// TIA Portal project "HBW" (V18)

(* hardware
DEVICE "S7-1200-Station_1"  S7-1200 Station
   slot 0: "Baugruppenträger_0"  S7-1200 Rack  Rack  V1.0
   slot 1: "HBW"  CPU 1215C DC/DC/DC  6ES7 215-1AG40-0XB0  V4.5
   slot 2: "DQ 8x24VDC _1"  SM 1222 DQ8 x 24VDC  6ES7 222-1BF32-0XB0  V2.0
*)

// ===== PLC "HBW"  CPU 1215C DC/DC/DC =====

VAR_GLOBAL   // PLC tag table "DrehSauger"
   "Schalter_sauger_oben" AT %I0.7 : Bool;
   "Schalter_sauger_mitte" AT %I1.0 : Bool;
   "Schalter_sauger_unten" AT %I1.1 : Bool;
   "ref_drehung" AT %I1.2 : Bool;
   "encoder_drehung_A" AT %I1.3 : Bool;
   "encoder_drehung_B" AT %I1.4 : Bool;
   "PWM_Drehbewegung" AT %QW1000 : Int;
   "drehung_counterclockwise" AT %Q8.2 : Bool;
   "drehung_clockwise" AT %Q8.3 : Bool;
   "Encoderwert_Drehbewegung" AT %ID1000 : DInt;
   "sauger_hoch" AT %Q8.0 : Bool;
   "sauger_runter" AT %Q8.1 : Bool;
   "ventil_vakuum" AT %Q8.4 : Bool;
   "kompressor" AT %Q8.5 : Bool;
   "Power_SaugerMotor" AT %Q1.1 : Bool;
END_VAR

VAR_GLOBAL   // PLC tag table "Hochregallager"
   "ref_HRL_Y" AT %I0.0 : Bool;
   "encoder_X_A" AT %I0.1 : Bool;
   "encoder_X_B" AT %I0.2 : Bool;
   "encoder_Y_A" AT %I0.3 : Bool;
   "encoder_Y_B" AT %I0.4 : Bool;
   "Schalter_RBG_vorn" AT %I0.5 : Bool;
   "Schalter_RBG_hinten" AT %I0.6 : Bool;
   "ref_hrl_X_horizontal" AT %I1.5 : Bool;
   "Encoderwert_X_Achse" AT %ID1004 : DInt;
   "Encoderwert_Y_Achse" AT %ID1008 : DInt;
   "xAchseZumRegal" AT %Q0.0 : Bool;
   "xAchseZumBand" AT %Q0.1 : Bool;
   "yAchseRunter" AT %Q0.2 : Bool;
   "yAchseHoch" AT %Q0.3 : Bool;
   "RBG_vor" AT %Q0.4 : Bool;
   "RBG_zurueck" AT %Q0.5 : Bool;
   "Power_RBG" AT %Q8.6 : Bool;
   "PWM_X_Achse" AT %QW1002 : Int;
   "PWM_Y_Achse" AT %QW1004 : Int;
END_VAR

DATA_BLOCK "DB_Global"   // DB2
{ S7_Optimized_Access := 'TRUE' }
VERSION : 0.1
   VAR
      DrehAchse : Struct
         referenziert : Bool;
      END_STRUCT;
      "X-Achse" : Struct
         referenziert : Bool;
      END_STRUCT;
      "Y-Achse" : Struct
         referenziert : Bool;
      END_STRUCT;
      RBG : Struct
         referenziert : Bool;
      END_STRUCT;
      Sauger : Struct
         referenziert : Bool;
      END_STRUCT;
      Order : Struct
         Pick : Struct
            pickAktiv : Bool;
            pickFinished : Bool;
            PICK : Bool;
            rack : String;
         END_STRUCT;
         Drop : Struct
            dropAktiv : Bool;
            dropFinished : Bool;
            DROP : Bool;
            rack : String;
         END_STRUCT;
         Park : Struct
            PARK : Bool;
            parkAktiv : Bool;
         END_STRUCT;
         Kalibriere : Struct
            kalibAktiv : Bool;
            KALIBRIERE : Bool;
            position_x : DInt;
            position_y : DInt;
            position_dreh : DInt;
            DEFAULT : Bool;
            defaultBeendet : Bool;
            ANFAHREN : Bool;
            anfahrenBeendet : Bool;
            BEENDEN : Bool;
            kalibriereFinished : Bool;
         END_STRUCT;
      END_STRUCT;
      Referenzieren : Bool;
      Referenziert : Bool;
      Busy : Bool;
   END_VAR
   VAR RETAIN
      RackPositionen : Struct
         A1 : Struct
            "type" : String;
            belegt : Bool;
            workpieceId : String;
         END_STRUCT;
         A2 : Struct
            "type" : String;
            belegt : Bool;
            workpieceId : String;
         END_STRUCT;
         A3 : Struct
            "type" : String;
            belegt : Bool;
            workpieceId : String;
         END_STRUCT;
         B1 : Struct
            "type" : String;
            belegt : Bool;
            workpieceId : String;
         END_STRUCT;
         B2 : Struct
            "type" : String;
            belegt : Bool;
            workpieceId : String;
         END_STRUCT;
         B3 : Struct
            "type" : String;
            belegt : Bool;
            workpieceId : String;
         END_STRUCT;
         C1 : Struct
            "type" : String;
            belegt : Bool;
            workpieceId : String;
         END_STRUCT;
         C2 : Struct
            "type" : String;
            belegt : Bool;
            workpieceId : String;
         END_STRUCT;
         C3 : Struct
            "type" : String;
            belegt : Bool;
            workpieceId : String;
         END_STRUCT;
      END_STRUCT;
      model : String := 'HBW';
   END_VAR
BEGIN
END_DATA_BLOCK

DATA_BLOCK "FB_DROP_DB"   // DB4
{ S7_Optimized_Access := 'TRUE' }
VERSION : 0.1
// stored: InstanceOfName FB_DROP
"FB_DROP"
BEGIN
END_DATA_BLOCK

DATA_BLOCK "FB_PICK_DB"   // DB5
{ S7_Optimized_Access := 'TRUE' }
VERSION : 0.1
// stored: InstanceOfName FB_PICK
"FB_PICK"
BEGIN
END_DATA_BLOCK

DATA_BLOCK "DB_Referenzen"   // DB7
{ S7_Optimized_Access := 'TRUE' }
VERSION : 0.1
   VAR RETAIN
      Calib : Struct
         "Y-Reihe" : Struct
            reihe_A : DInt := 80;
            reihe_B : DInt := 430;
            reihe_C : DInt := 825;
            Offset : DInt := 60;
         END_STRUCT;
         Park : Struct
            position_x : DInt := 1100;
            position_y : DInt := 825;
            position_dreh : DInt := 450;
         END_STRUCT;
         "X-Spalte" : Struct
            spalte_1 : DInt := 715;
            spalte_2 : DInt := 1300;
            spalte_3 : DInt := 1888;
         END_STRUCT;
         Rampe : Struct
            position_X : DInt := 248;
            position_Y : DInt := 600;
            position_dreh : DInt := 630;
            position_drehCheck : DInt := 450;
            offset : DInt := 220;
         END_STRUCT;
         FTS : Struct
            Dreh : DInt := 29;
         END_STRUCT;
         Limits : Struct
            grenze_x_oben : DInt := 2000;
            grenze_x_unten : DInt := 0;
            grenze_y_oben : DInt := 820;
            grenze_y_unten : DInt := 0;
            grenze_dreh_oben : DInt := 650;
            grenze_dreh_unten : DInt := 0;
         END_STRUCT;
         Zeiten : Struct
            zeit_prozessende : Time := T#2S;
            zeit_saugerVentilAuf : Time := T#1S;
            zeit_saugerVentilZu : Time := T#500MS;
            zeit_kompressor : Time := T#1S;
         END_STRUCT;
      END_STRUCT;
      Defaults : Struct
         "Y-Reihe" : Struct
            reihe_A : DInt := 80;
            reihe_B : DInt := 430;
            reihe_C : DInt := 825;
            Offset : DInt := 60;
         END_STRUCT;
         Park : Struct
            position_x : DInt;
            position_y : DInt;
            position_dreh : DInt;
         END_STRUCT;
         "X-Spalte" : Struct
            spalte_1 : DInt := 715;
            spalte_2 : DInt := 1300;
            spalte_3 : DInt := 1888;
         END_STRUCT;
         Rampe : Struct
            position_X : DInt := 248;
            position_Y : DInt := 600;
            position_dreh : DInt := 630;
            position_drehCheck : DInt := 450;
            offset : DInt := 220;
         END_STRUCT;
         FTS : Struct
            Dreh : DInt := 29;
         END_STRUCT;
         Limits : Struct
            grenze_x_oben : DInt := 2000;
            grenze_x_unten : DInt := 0;
            grenze_y_oben : DInt := 820;
            grenze_y_unten : DInt := 0;
            grenze_dreh_oben : DInt := 650;
            grenze_dreh_unten : DInt := 0;
         END_STRUCT;
         Zeiten : Struct
            zeit_prozessende : Time := T#2S;
            zeit_saugerVentilAuf : Time := T#1S;
            zeit_saugerVentilZu : Time := T#500MS;
            zeit_kompressor : Time := T#1S;
         END_STRUCT;
      END_STRUCT;
      PWM_schnell : DInt := 100;
      PWM_langsam : DInt := 50;
      range : DInt := 1;
      slowRange : DInt := 25;
   END_VAR
BEGIN
END_DATA_BLOCK

DATA_BLOCK "FB_OrderOrganisation_DB"   // DB8
{ S7_Optimized_Access := 'TRUE' }
VERSION : 0.1
// stored: InstanceOfName FB_OrderOrganisation
"FB_OrderOrganisation"
BEGIN
END_DATA_BLOCK

DATA_BLOCK "DB_Version"   // DB9
TITLE = Version
{ S7_Optimized_Access := 'TRUE' }
VERSION : 0.1
   VAR RETAIN
      "version" : String := '1.0.1';   // Versionierung
   END_VAR
BEGIN
END_DATA_BLOCK

DATA_BLOCK "FB_KALIBRIERE_DB"   // DB10
{ S7_Optimized_Access := 'TRUE' }
VERSION : 0.1
// stored: InstanceOfName FB_KALIBRIERE
"FB_KALIBRIERE"
BEGIN
END_DATA_BLOCK

// folder: EncoderMoves

DATA_BLOCK "FB_Positionierung_DB"   // DB15
{ S7_Optimized_Access := 'TRUE' }
VERSION : 0.1
// stored: InstanceOfName FB_Positionierung
"FB_Positionierung"
BEGIN
END_DATA_BLOCK

// folder: (top level)

FUNCTION_BLOCK "FB_PICK"   // FB2, FBD
{ S7_Optimized_Access := 'TRUE' }
VERSION : 0.1
   VAR
      Positionen : Struct
         Rack : Struct
            position_X : DInt;
            position_Y : DInt;
            position_Y_mitOffset : DInt;
         END_STRUCT;
         Rampe : Struct
            position_X : DInt;
            position_Y : DInt;
            position_Y_mitOffset : DInt;
            position_dreh : DInt;
            position_drehCheck : DInt;
         END_STRUCT;
         FTS : Struct
            position_dreh : DInt;
         END_STRUCT;
      END_STRUCT;
      zielRack : Struct
         Position_X : DInt;
         Position_Y : DInt;
      END_STRUCT;
      start : Bool;
      busyPick : Bool;
      "step" : DInt;
      stepSauger : DInt;
      finished : Bool;
      Sauger : Struct
         busy : Bool;
         aufDrehCheck : Bool;
      END_STRUCT;
      Lager : Struct
         stepLager : DInt;
         busy : Bool;
         aufRampe : Bool;
      END_STRUCT;
      warteHaupt : TON_TIME;
      warteHauptStart : Bool;
      warteHauptTime : Time := T#300MS;
      warteNeben : TON_TIME;
      warteNebenStart : Bool;
      warteNebenTime : Time := T#1s;
   END_VAR
BEGIN

REGION Network 1: Zeiten
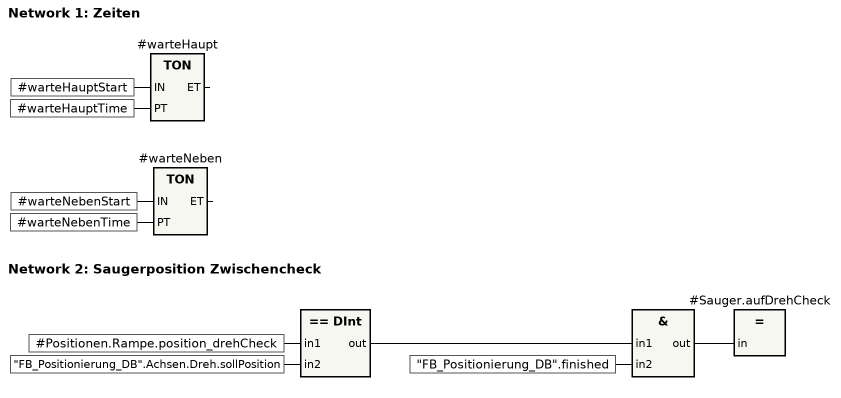
   #warteHaupt(IN := #warteHauptStart, PT := #warteHauptTime);   // TON
   #warteNeben(IN := #warteNebenStart, PT := #warteNebenTime);   // TON
END_REGION

REGION Network 2: Saugerposition Zwischencheck
   #Sauger.aufDrehCheck := (#Positionen.Rampe.position_drehCheck = "FB_Positionierung_DB".Achsen.Dreh.sollPosition) AND "FB_Positionierung_DB".finished;
END_REGION

REGION Network 3 (SCL): Grundlegender Ablauf von PICK
   CASE #step OF
       0: // Init
           IF #start  THEN
               #start := FALSE;

               // Motoren An
               "Power_SaugerMotor" := TRUE;
               "Power_RBG" := TRUE;

               // Positionen Rack laden
               #Positionen.Rack.position_X := #zielRack.Position_X;
               #Positionen.Rack.position_Y := #zielRack.Position_Y;
               #Positionen.Rack.position_Y_mitOffset := #zielRack.Position_Y - "DB_Referenzen".Calib."Y-Reihe".Offset;

               // Positionen Rampe laden
               #Positionen.Rampe.position_X := "DB_Referenzen".Calib.Rampe.position_X;
               #Positionen.Rampe.position_Y := "DB_Referenzen".Calib.Rampe.position_Y;
               #Positionen.Rampe.position_Y_mitOffset := "DB_Referenzen".Calib.Rampe.position_Y + "DB_Referenzen".Calib.Rampe.offset;
               #Positionen.Rampe.position_dreh := "DB_Referenzen".Calib.Rampe.position_dreh;
               #Positionen.Rampe.position_drehCheck := "DB_Referenzen".Calib.Rampe.position_drehCheck;

               // Positionen FTS laden
               #Positionen.FTS.position_dreh := "DB_Referenzen".Calib.FTS.Dreh;

               // busy 
               #step := 10;
           END_IF
           ;
       10: // Starte PICK
           // Rack anfahren

           // Positionen übergeben
           "FB_Positionierung_DB".Achsen.X.sollPosition := #Positionen.Rack.position_X;
           "FB_Positionierung_DB".Achsen.Y.sollPosition := #Positionen.Rack.position_Y;
           "FB_Positionierung_DB".Achsen.Dreh.sollPosition := #Positionen.FTS.position_dreh;

           // Start der Positionierung
           "FB_Positionierung_DB".finished := FALSE;
           "FB_Positionierung_DB".startPositionierung := TRUE;
           #step := 11
           ;
       11: // Ende Positionierung
           IF "FB_Positionierung_DB".finished THEN
               #step := 20;
           END_IF
           ;
       20: // Starte Paralleles Netzwerke um Workpiece zu holen
           IF #stepSauger = 0 THEN
               #stepSauger := 1;
               #step := 25;
           END_IF
           ;
       25: // RBG rausfahren

           // RBG unter Container fahren
           "RBG_vor" := TRUE;
           "RBG_zurueck" := FALSE;
           IF "Schalter_RBG_vorn" AND NOT "Schalter_RBG_hinten" THEN
               "RBG_vor" := FALSE;
               "RBG_zurueck" := FALSE;
               #step := 30;
           END_IF
           ;
       30: // Container anheben
           // Position übergeben und starten
           "FB_Positionierung_DB".Achsen.Y.sollPosition := #Positionen.Rack.position_Y_mitOffset;
           "FB_Positionierung_DB".finished := FALSE;
           "FB_Positionierung_DB".startPositionierung := TRUE;
           #step := 31
           ;
       31: // Ende Positionierung
           IF "FB_Positionierung_DB".finished THEN
               #step := 35;
           END_IF
           ;
       35: // RBG rein
           "RBG_vor" := FALSE;
           "RBG_zurueck" := TRUE;
           IF "Schalter_RBG_hinten" AND NOT "Schalter_RBG_vorn" THEN
               "RBG_vor" := FALSE;
               "RBG_zurueck" := FALSE;
               #step := 40;
           END_IF
           ;
       40: // Zur Rampe
           // Positionen übergeben und starten
           "FB_Positionierung_DB".Achsen.X.sollPosition := #Positionen.Rampe.position_X;
           "FB_Positionierung_DB".Achsen.Y.sollPosition := #Positionen.Rampe.position_Y;
           "FB_Positionierung_DB".finished := FALSE;
           "FB_Positionierung_DB".startPositionierung := TRUE;
           #step := 41
           ;
       41: // Ende Positionerung
           IF "FB_Positionierung_DB".finished THEN
               #step := 45;
           END_IF
           ;
       45: // RBG raus
           "RBG_vor" := TRUE;
           "RBG_zurueck" := FALSE;
           IF "Schalter_RBG_vorn" AND NOT "Schalter_RBG_hinten" THEN
               "RBG_vor" := FALSE;
               "RBG_zurueck" := FALSE;
               #step := 50;
           END_IF
           ;
       50: // Container auf Rampe ablegen
           "FB_Positionierung_DB".Achsen.Y.sollPosition := #Positionen.Rampe.position_Y_mitOffset;
           "FB_Positionierung_DB".finished := FALSE;
           "FB_Positionierung_DB".startPositionierung := TRUE;
           #step := 51
           ;
       51: // Ende Positionierung
           IF "FB_Positionierung_DB".finished THEN
               #step := 60;
           END_IF
           ;
       60: // Check ob Drehachse auf position
           IF #Sauger.aufDrehCheck THEN
               #step := 61;
           END_IF
           ;
       61: // Dreh Achse über Rampe fahren
           "FB_Positionierung_DB".Achsen.Dreh.sollPosition := #Positionen.Rampe.position_dreh;
           "FB_Positionierung_DB".finished := FALSE;
           "FB_Positionierung_DB".startPositionierung := TRUE;
           #step := 62
           ;
       62: // Ende Positionierung
           IF "FB_Positionierung_DB".finished THEN
               #step := 70;
           END_IF
           ;
       70: // Sauger runter bis Schalter Mitte
           "sauger_runter" := TRUE;
           "sauger_hoch" := FALSE;
           IF "Schalter_sauger_mitte" THEN
               "sauger_runter" := FALSE;
               "sauger_hoch" := FALSE;
               #step := 71;
           END_IF
           ;
       71: // ventil lösen
           "ventil_vakuum" := FALSE;
           "kompressor" := FALSE;
           #warteHauptTime := "DB_Referenzen".Calib.Zeiten.zeit_saugerVentilAuf;
           #warteHauptStart := TRUE;
           IF #warteHaupt.Q THEN
               #warteHauptStart := FALSE;
               #step := 72;
           END_IF
           ;
       72: // Sauger nach oben
           "sauger_runter" := FALSE;
           "sauger_hoch" := TRUE;
           IF "Schalter_sauger_oben" THEN
               "sauger_runter" := FALSE;
               "sauger_hoch" := FALSE;
               #step := 73;
           END_IF
           ;
       73: // DrehAchse auf CheckPosition
           "FB_Positionierung_DB".Achsen.Dreh.sollPosition := #Positionen.Rampe.position_drehCheck;
           "FB_Positionierung_DB".finished := FALSE;
           "FB_Positionierung_DB".startPositionierung := TRUE;
           #step := 74
           ;
           74: // Ende Positionierung
           IF "FB_Positionierung_DB".finished THEN
               #step := 75;
           END_IF
           ;
       75: // Container anheben
           "FB_Positionierung_DB".Achsen.Y.sollPosition := #Positionen.Rampe.position_Y;
           "FB_Positionierung_DB".finished := FALSE;
           "FB_Positionierung_DB".startPositionierung := TRUE;
           #step := 76;
       76: // Ende Positionierung
           IF "FB_Positionierung_DB".finished THEN
               #step := 80;
           END_IF
           ;
       80: // RBG rein
           "RBG_vor" := FALSE;
           "RBG_zurueck" := TRUE;
           IF "Schalter_RBG_hinten" THEN
               "RBG_vor" := FALSE;
               "RBG_zurueck" := FALSE;
               #step := 85;
           END_IF
           ;
       85: // Auf Rack position und FTS Position Fahren
           "FB_Positionierung_DB".Achsen.X.sollPosition := #Positionen.Rack.position_X;
           "FB_Positionierung_DB".Achsen.Y.sollPosition := #Positionen.Rack.position_Y_mitOffset;
           "FB_Positionierung_DB".Achsen.Dreh.sollPosition := #Positionen.FTS.position_dreh;

           "FB_Positionierung_DB".finished := FALSE;
           "FB_Positionierung_DB".startPositionierung := TRUE;
           #step := 86
           ;
           86: // Ende Positionierung
           IF "FB_Positionierung_DB".finished THEN
               #step := 90;
           END_IF
           ;
       90: // RBG raus
           "RBG_vor" := TRUE;
           "RBG_zurueck" := FALSE;
           IF "Schalter_RBG_vorn" THEN
               "RBG_vor" := FALSE;
               "RBG_zurueck" := FALSE;
               #step := 91;
           END_IF
           ;
       91: // Container ablegen 
           "FB_Positionierung_DB".Achsen.Y.sollPosition := #Positionen.Rack.position_Y;
           "FB_Positionierung_DB".finished := FALSE;
           "FB_Positionierung_DB".startPositionierung := TRUE;
           #step := 92
           ;
       92: // Ende Positionierung
           IF "FB_Positionierung_DB".finished THEN
               #step := 95;
           END_IF
           ;
       95: // RBG rein
           "RBG_vor" := FALSE;
           "RBG_zurueck" := TRUE;
           IF "Schalter_RBG_hinten" AND NOT "Schalter_RBG_vorn" THEN
               "RBG_vor" := FALSE;
               "RBG_zurueck" := FALSE;
               #step := 100;
           END_IF
           ;
       100: // ENDE
           "Power_SaugerMotor" := FALSE;
           "Power_RBG" := FALSE;
           #finished := TRUE;
           #warteHauptTime := T#200ms;
           #warteHauptStart := TRUE;
           IF #warteHaupt.Q THEN
               #warteHauptStart := FALSE;
               #step := 0;
           END_IF
           ;

       ELSE  // Statement section ELSE
           ;
   END_CASE;
END_REGION

REGION Network 4 (SCL): Worpiece vom FTS holen
   CASE #stepSauger OF
       0: // Wartet auf Externe Eingabe
           #Sauger.busy := FALSE
           ;
       1:  // busy
           #Sauger.busy := TRUE;
           #stepSauger := 10
           ;
       10: // Sauger runter bis Schalter unten
           "sauger_runter" := TRUE;
           "sauger_hoch" := FALSE;
           IF "Schalter_sauger_unten" THEN
               "sauger_runter" := FALSE;
               "sauger_hoch" := FALSE;
               #stepSauger := 20;
           END_IF
           ;
       20: // kompressor an
           "kompressor" := TRUE;
           #warteNebenTime := "DB_Referenzen".Calib.Zeiten.zeit_kompressor;
           #warteNebenStart := TRUE;
           IF #warteNeben.Q THEN
               #warteNebenStart := FALSE;
               #stepSauger := 30;
           END_IF
           ;
       30: // ventil zumachen
           "ventil_vakuum" := TRUE;
           #stepSauger := 40
           ;
       40: // kompressor aus und hoch bis schalter oben
           "sauger_runter" := FALSE;
           "sauger_hoch" := TRUE;
           IF "Schalter_sauger_oben" THEN
               "sauger_runter" := FALSE;
               "sauger_hoch" := FALSE;
               #stepSauger := 50;
           END_IF
           ;
       50: // Position an Positionierung senden
           "FB_Positionierung_DB".Achsen.Dreh.sollPosition := #Positionen.Rampe.position_drehCheck;
           #stepSauger := 60
           ;
       60: // finished
           #stepSauger := 0;
           ;
           ELSE  // Statement section ELSE
               ;
   END_CASE;
END_REGION
END_FUNCTION_BLOCK

FUNCTION_BLOCK "FB_DROP"   // FB3, FBD
{ S7_Optimized_Access := 'TRUE' }
VERSION : 0.1
   VAR
      Positionen : Struct
         Rack : Struct
            position_X : DInt;
            position_Y : DInt;
            position_Y_mitOffset : DInt;
         END_STRUCT;
         Rampe : Struct
            position_X : DInt;
            position_Y : DInt;
            position_Y_mitOffset : DInt;
            position_dreh : DInt;
            position_drehCheck : DInt;
         END_STRUCT;
         FTS : Struct
            position_dreh : DInt;
         END_STRUCT;
      END_STRUCT;
      zielRack : Struct
         Position_X : DInt;
         Position_Y : DInt;
      END_STRUCT;
      start : Bool;
      busyDrop : Bool;
      "step" : DInt;
      stepSauger : DInt;
      finished : Bool;
      warteHaupt : TON_TIME;
      warteHauptStart : Bool;
      warteHauptTime : Time := T#300MS;
      warteNeben : TON_TIME;
      warteNebenStart : Bool;
      warteNebenTime : Time := T#1s;
   END_VAR
BEGIN

REGION Network 1 (SCL): Drop Ablauf
   CASE #step OF

       0: // --------------- Init

           IF #start THEN

               #start := FALSE;

               // Motoren an
               "Power_RBG" := TRUE;
               "Power_SaugerMotor" := TRUE;

               // Positionen Rack laden
               #Positionen.Rack.position_X := #zielRack.Position_X;
               #Positionen.Rack.position_Y := #zielRack.Position_Y;
               #Positionen.Rack.position_Y_mitOffset := #zielRack.Position_Y - "DB_Referenzen".Calib."Y-Reihe".Offset;

               // Positionen Rampe laden
               #Positionen.Rampe.position_X := "DB_Referenzen".Calib.Rampe.position_X;
               #Positionen.Rampe.position_Y := "DB_Referenzen".Calib.Rampe.position_Y;
               #Positionen.Rampe.position_Y_mitOffset := "DB_Referenzen".Calib.Rampe.position_Y + "DB_Referenzen".Calib.Rampe.offset;
               #Positionen.Rampe.position_dreh := "DB_Referenzen".Calib.Rampe.position_dreh;
               #Positionen.Rampe.position_drehCheck := "DB_Referenzen".Calib.Rampe.position_drehCheck;

               // Positionen FTS laden
               #Positionen.FTS.position_dreh := "DB_Referenzen".Calib.FTS.Dreh;

               #step := 9;
           END_IF
           ;
       9: // --------------- Ausgansposition
           "sauger_hoch" := TRUE;
           "sauger_runter" := FALSE;
           IF "Schalter_sauger_oben" THEN
               "sauger_hoch" := FALSE;
               "sauger_runter" := FALSE;
               #step := 10;
           END_IF
           ;
       10: // --------------- --------------- Starte Drop



           // Positionen übertragen
           "FB_Positionierung_DB".Achsen.X.sollPosition := #Positionen.Rack.position_X;
           "FB_Positionierung_DB".Achsen.Y.sollPosition := #Positionen.Rack.position_Y;
           "FB_Positionierung_DB".Achsen.Dreh.sollPosition := #Positionen.Rampe.position_drehCheck;

           // Start positionerung
           "FB_Positionierung_DB".finished := FALSE;
           "FB_Positionierung_DB".startPositionierung := TRUE;
           #step := 11
           ;
       11: // --------------- Ende Positionierung
           IF "FB_Positionierung_DB".finished THEN
               #step := 20;
           END_IF
           ;
       20: // --------------- RBG rausfahren unter Container
           "RBG_vor" := TRUE;
           "RBG_zurueck" := FALSE;
           IF "Schalter_RBG_vorn" AND NOT "Schalter_RBG_hinten" THEN
               "RBG_vor" := FALSE;
               "RBG_zurueck" := FALSE;
               #step := 30;
           END_IF
           ;
       30: // --------------- Container anheben

           // Positionen übertragen
           "FB_Positionierung_DB".Achsen.Y.sollPosition := #Positionen.Rack.position_Y_mitOffset;

           // Start Positionierung
           "FB_Positionierung_DB".finished := FALSE;
           "FB_Positionierung_DB".startPositionierung := TRUE;

           #step := 31
           ;
       31: // --------------- Ende Positionierung
           IF "FB_Positionierung_DB".finished THEN
               #step := 40;
           END_IF
           ;
       40: // --------------- RBG reinfahren
           "RBG_vor" := FALSE;
           "RBG_zurueck" := TRUE;
           IF "Schalter_RBG_hinten" AND NOT "Schalter_RBG_vorn" THEN
               "RBG_vor" := FALSE;
               "RBG_zurueck" := FALSE;
               #step := 50;
           END_IF
           ;
       50: // --------------- Zur Rampe

           // Positionen übertragen
           "FB_Positionierung_DB".Achsen.X.sollPosition := #Positionen.Rampe.position_X;
           "FB_Positionierung_DB".Achsen.Y.sollPosition := #Positionen.Rampe.position_Y;

           // Positionierung starten
           "FB_Positionierung_DB".finished := FALSE;
           "FB_Positionierung_DB".startPositionierung := TRUE;
           #step := 51
           ;
       51: // --------------- Ende Positionierung
           IF "FB_Positionierung_DB".finished THEN
               #step := 60;
           END_IF
           ;
       60: // --------------- RBG raus
           "RBG_vor" := TRUE;
           "RBG_zurueck" := FALSE;
           IF "Schalter_RBG_vorn" AND NOT "Schalter_RBG_hinten" THEN
               "RBG_vor" := FALSE;
               "RBG_zurueck" := FALSE;
               #step := 70;
           END_IF
           ;
       70: // --------------- Container ablegen -- Rampe mit Offset

           // Positionen übertragen
           "FB_Positionierung_DB".Achsen.Y.sollPosition := #Positionen.Rampe.position_Y_mitOffset;

           // Start positionierung
           "FB_Positionierung_DB".finished := FALSE;
           "FB_Positionierung_DB".startPositionierung := TRUE;
           #step := 71
           ;
       71: // --------------- Ende Positionierung
           IF "FB_Positionierung_DB".finished THEN
               #step := 80;
           END_IF
           ;
       80: // --------------- Sauger auf Position Rampe

           // Positionen übertragen
           "FB_Positionierung_DB".Achsen.Dreh.sollPosition := #Positionen.Rampe.position_dreh;

           // Start positionierung
           "FB_Positionierung_DB".finished := FALSE;
           "FB_Positionierung_DB".startPositionierung := TRUE;
           #step := 81
           ;

       81: // --------------- Ende Positionierung
           IF "FB_Positionierung_DB".finished THEN
               #step := 90;
           END_IF
           ;
       90: // --------------- Sauger runter bis Schalter mitte
           "sauger_runter" := TRUE;
           "sauger_hoch" := FALSE;
           IF "Schalter_sauger_mitte" THEN
               "sauger_runter" := FALSE;
               "sauger_hoch" := FALSE;
               #step := 91;
           END_IF
           ;
       91: // --------------- Kompressor an
           "kompressor" := TRUE;
           #warteHauptTime := "DB_Referenzen".Calib.Zeiten.zeit_kompressor;
           #warteHauptStart := TRUE;
           IF #warteHaupt.Q THEN
               #warteHauptStart := FALSE;
               #step := 92;
           END_IF
           ;
       92: // --------------- ventil zu
           "ventil_vakuum" := TRUE;
           #warteHauptTime := "DB_Referenzen".Calib.Zeiten.zeit_saugerVentilZu;
           #warteHauptStart := TRUE;
           IF #warteHaupt.Q THEN
               #warteHauptStart := FALSE;
               #step := 93;
           END_IF
           ;
       93: // --------------- sauger hoch bis schalter oben
           "sauger_runter" := FALSE;
           "sauger_hoch" := TRUE;
           IF "Schalter_sauger_oben" THEN
               "sauger_runter" := FALSE;
               "sauger_hoch" := FALSE;
               #step := 100;
           END_IF
           ;
       100: // --------------- Zwischenposition anfahren

           // Positionen übertragen
           "FB_Positionierung_DB".Achsen.Dreh.sollPosition := #Positionen.Rampe.position_drehCheck;

           // Start Positionierung
           "FB_Positionierung_DB".finished := FALSE;
           "FB_Positionierung_DB".startPositionierung := TRUE;
           #step := 101
           ;
       101: // --------------- Ende Positionierung
           IF "FB_Positionierung_DB".finished THEN
               #step := 110;
           END_IF
           ;
       110: // --------------- Container anheben und FTS Position anfahren

           // Positionen übertragen
           "FB_Positionierung_DB".Achsen.Y.sollPosition := #Positionen.Rampe.position_Y;
           "FB_Positionierung_DB".Achsen.Dreh.sollPosition := #Positionen.FTS.position_dreh;

           // Start Positionierung
           "FB_Positionierung_DB".finished := FALSE;
           "FB_Positionierung_DB".startPositionierung := TRUE;
           #step := 111
           ;
       111: // --------------- Ende Positionierung
           IF "FB_Positionierung_DB".finished THEN
               #step := 112;
           END_IF
           ;
       112: // --------------- Starte Parallel Netzwerk
           #stepSauger := 1;
           #step := 120
           ;
       120: // --------------- RBG rein
           "RBG_vor" := FALSE;
           "RBG_zurueck" := TRUE;
           IF NOT "Schalter_RBG_vorn" AND "Schalter_RBG_hinten" THEN
               "RBG_vor" := FALSE;
               "RBG_zurueck" := FALSE;
               #step := 130;
           END_IF
           ;
       130: // --------------- Rack Position anfahren mit Offset

           // Positionen übertragen
           "FB_Positionierung_DB".Achsen.X.sollPosition := #Positionen.Rack.position_X;
           "FB_Positionierung_DB".Achsen.Y.sollPosition := #Positionen.Rack.position_Y_mitOffset;

           // Start Positionierung
           "FB_Positionierung_DB".finished := FALSE;
           "FB_Positionierung_DB".startPositionierung := TRUE;
           #step := 131
           ;
       131: // --------------- Ende Positionierung
           IF "FB_Positionierung_DB".finished THEN
               #step := 140;
           END_IF
           ;
       140: // --------------- RBG raus
           "RBG_vor" := TRUE;
           "RBG_zurueck" := FALSE;
           IF "Schalter_RBG_vorn" AND NOT "Schalter_RBG_hinten" THEN
               "RBG_vor" := FALSE;
               "RBG_zurueck" := FALSE;
               #step := 150;
           END_IF
           ;
       150: // --------------- Container abstellen

           // Positionen übertragen
           "FB_Positionierung_DB".Achsen.Y.sollPosition := #Positionen.Rack.position_Y;

           // Start Positionierung
           "FB_Positionierung_DB".finished := FALSE;
           "FB_Positionierung_DB".startPositionierung := TRUE;
           #step := 151
           ;
       151: // --------------- Ende Positionierung
           IF "FB_Positionierung_DB".finished THEN
               #step := 160;
           END_IF
           ;
       160: // --------------- RBG rein
           "RBG_vor" := FALSE;
           "RBG_zurueck" := TRUE;
           IF NOT "Schalter_RBG_vorn" AND  "Schalter_RBG_hinten" THEN
               "RBG_vor" := FALSE;
               "RBG_zurueck" := FALSE;
               #step := 170;
           END_IF
           ;
       170: // Check ob Sauger fertig
           IF #stepSauger = 100 THEN
               #stepSauger := 0;
               #step := 200;
           END_IF
           ;
       200: // --------------- ENDE
           // Motoren an
           "Power_RBG" := FALSE;
           "Power_SaugerMotor" := FALSE;
           #finished := TRUE;
           #step := 0;
       ELSE  // Statement section ELSE
           ;
   END_CASE;
END_REGION

REGION Network 2 (SCL): Parallel Zusatz
   CASE #stepSauger OF
       0: // Warte auf Aktivierung
           ;
       1: // Starte Drop auf FTS
           "sauger_runter" := TRUE;
           "sauger_hoch" := FALSE;
           IF "Schalter_sauger_unten" THEN
               "sauger_runter" := FALSE;
               "sauger_hoch" := FALSE;
               #stepSauger := 20;
           END_IF
           ;
       20: // Ventil lösen und kompressor aus
           "kompressor" := FALSE;
           "ventil_vakuum" := FALSE;
           #warteNebenTime := "DB_Referenzen".Calib.Zeiten.zeit_saugerVentilAuf;
           #warteNebenStart := TRUE;
           IF #warteNeben.Q THEN
               #warteNebenStart := FALSE;
               #stepSauger := 30;
           END_IF
           ;
       30: // Sauger hoch bis schalter oben
           "sauger_runter" := FALSE;
           "sauger_hoch" := TRUE;
           IF "Schalter_sauger_oben" THEN
               "sauger_runter" := FALSE;
               "sauger_hoch" := FALSE;
               #stepSauger := 100;
           END_IF
           ;
       100: // warte auf reset

           ;
       ELSE  // Statement section ELSE
           ;
   END_CASE;
END_REGION

REGION Network 3: Zeiten
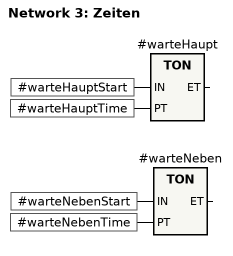
   #warteHaupt(IN := #warteHauptStart, PT := #warteHauptTime);   // TON
   #warteNeben(IN := #warteNebenStart, PT := #warteNebenTime);   // TON
END_REGION
END_FUNCTION_BLOCK

FUNCTION_BLOCK "FB_OrderOrganisation"   // FB4, FBD
{ S7_Optimized_Access := 'TRUE' }
VERSION : 0.1
   VAR
      "step" : DInt;
      warte : TON_TIME;
      warteStart : Bool;
      warteZeit : Time;
   END_VAR
BEGIN

REGION Network 1: Zeiten
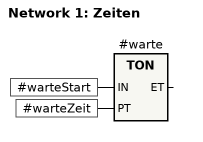
   #warte(IN := #warteStart, PT := #warteZeit);   // TON
END_REGION

REGION Network 2 (SCL): Ablauf
   CASE #step OF
       0:  // Init
           IF NOT "DB_Global".Busy THEN
               #step := 1;
           END_IF
           ;

       1: // OrderManagement
           IF "DB_Global".Order.Kalibriere.KALIBRIERE THEN
               // HBW Status setzen
               "DB_Global".Order.Kalibriere.kalibAktiv := TRUE;
               "DB_Global".Order.Kalibriere.KALIBRIERE := FALSE;
               #step := 10;
           ELSIF "DB_Global".Order.Pick.PICK THEN
               // HBW Status setzen
               "DB_Global".Order.Pick.pickAktiv := TRUE;
               "DB_Global".Order.Pick.PICK := FALSE;
               #step := 20;
           ELSIF "DB_Global".Order.Drop.DROP THEN
               // HBW Status setzen
               "DB_Global".Order.Drop.dropAktiv := TRUE;
               "DB_Global".Order.Drop.DROP := FALSE;
               #step := 30;
           END_IF
           ;
       200: // Ende für jeden Prozess
           #warteZeit := "DB_Referenzen".Calib.Zeiten.zeit_prozessende;
           #warteStart := TRUE;
           IF #warte.Q THEN
               #warteStart := FALSE;
               "DB_Global".Order.Pick.pickFinished := FALSE;
               "DB_Global".Order.Drop.dropFinished := FALSE;
               "DB_Global".Order.Kalibriere.kalibriereFinished := FALSE;
               #step := 0;
           END_IF
           ;
       10: // Starte Kalibrierung
           #step := 11
           ;
       11: // warte auf Ende Kalibrierung
           IF "FB_KALIBRIERE_DB".fertig THEN
               #step := 12;
           END_IF
           ;
       12: // starte Referenzierung
           "DB_Global".DrehAchse.referenziert := FALSE;
           "DB_Global"."X-Achse".referenziert := FALSE;
           "DB_Global"."Y-Achse".referenziert := FALSE;
           IF "DB_Global".Referenziert THEN
               #step := 13;
           END_IF
           ;
       13: // setzte Finished Flag
           "DB_Global".Order.Kalibriere.kalibriereFinished := TRUE;
           "DB_Global".Order.Kalibriere.kalibAktiv := FALSE;
           #step := 200;

           // -------------------- ENDE Kalibrierung -------------------- 
           // 
       20: // PICK Zielposition übertragen

           // Zielposition übergeben
           IF "DB_Global".Order.Pick.rack = 'A1' THEN
               "FB_PICK_DB".zielRack.Position_Y := "DB_Referenzen".Calib."Y-Reihe".reihe_A;
               "FB_PICK_DB".zielRack.Position_X := "DB_Referenzen".Calib."X-Spalte".spalte_1;

           ELSIF "DB_Global".Order.Pick.rack = 'A2' THEN
               "FB_PICK_DB".zielRack.Position_Y := "DB_Referenzen".Calib."Y-Reihe".reihe_A;
               "FB_PICK_DB".zielRack.Position_X := "DB_Referenzen".Calib."X-Spalte".spalte_2;

           ELSIF "DB_Global".Order.Pick.rack = 'A3' THEN
               "FB_PICK_DB".zielRack.Position_Y := "DB_Referenzen".Calib."Y-Reihe".reihe_A;
               "FB_PICK_DB".zielRack.Position_X := "DB_Referenzen".Calib."X-Spalte".spalte_3;

           ELSIF "DB_Global".Order.Pick.rack = 'B1' THEN
               "FB_PICK_DB".zielRack.Position_Y := "DB_Referenzen".Calib."Y-Reihe".reihe_B;
               "FB_PICK_DB".zielRack.Position_X := "DB_Referenzen".Calib."X-Spalte".spalte_1;

           ELSIF "DB_Global".Order.Pick.rack = 'B2' THEN
               "FB_PICK_DB".zielRack.Position_Y := "DB_Referenzen".Calib."Y-Reihe".reihe_B;
               "FB_PICK_DB".zielRack.Position_X := "DB_Referenzen".Calib."X-Spalte".spalte_2;

           ELSIF "DB_Global".Order.Pick.rack = 'B3' THEN
               "FB_PICK_DB".zielRack.Position_Y := "DB_Referenzen".Calib."Y-Reihe".reihe_B;
               "FB_PICK_DB".zielRack.Position_X := "DB_Referenzen".Calib."X-Spalte".spalte_3;

           ELSIF "DB_Global".Order.Pick.rack = 'C1' THEN
               "FB_PICK_DB".zielRack.Position_Y := "DB_Referenzen".Calib."Y-Reihe".reihe_C;
               "FB_PICK_DB".zielRack.Position_X := "DB_Referenzen".Calib."X-Spalte".spalte_1;

           ELSIF "DB_Global".Order.Pick.rack = 'C2' THEN
               "FB_PICK_DB".zielRack.Position_Y := "DB_Referenzen".Calib."Y-Reihe".reihe_C;
               "FB_PICK_DB".zielRack.Position_X := "DB_Referenzen".Calib."X-Spalte".spalte_2;

           ELSIF "DB_Global".Order.Pick.rack = 'C3' THEN
               "FB_PICK_DB".zielRack.Position_Y := "DB_Referenzen".Calib."Y-Reihe".reihe_C;
               "FB_PICK_DB".zielRack.Position_X := "DB_Referenzen".Calib."X-Spalte".spalte_3;

           END_IF
           ;
           #step := 21
           ;
       21: // Starte Pick Process
           "FB_PICK_DB".finished := FALSE;
           "FB_PICK_DB".start := TRUE;
           #step := 22
           ;
       22: // Warte auf Finish
           IF "FB_PICK_DB".finished THEN
               #step := 23;
           END_IF
           ;

       23: // referenzieren
           "DB_Global".DrehAchse.referenziert := FALSE;
           "DB_Global"."X-Achse".referenziert := FALSE;
           "DB_Global"."Y-Achse".referenziert := FALSE;
           #step := 24
           ;
       24: // warte auf Referenzierung
           IF "DB_Global".Referenziert THEN
               #step := 25;
           END_IF
           ;
       25: // bestätige erfolgreichen Abschluss 
           "DB_Global".Order.Pick.pickFinished := TRUE;
           "DB_Global".Order.Pick.pickAktiv := FALSE;
           "FB_PICK_DB".finished := FALSE;
           #step := 200
           ;
           // -------------------- ENDE PICK --------------------

       30: // DROP Zielposition übertragen
           // Zielposition übergeben
           IF "DB_Global".Order.Drop.rack = 'A1' THEN
               "FB_DROP_DB".zielRack.Position_X := "DB_Referenzen".Calib."X-Spalte".spalte_1;
               "FB_DROP_DB".zielRack.Position_Y := "DB_Referenzen".Calib."Y-Reihe".reihe_A;
           ELSIF "DB_Global".Order.Drop.rack = 'A2' THEN
               "FB_DROP_DB".zielRack.Position_X := "DB_Referenzen".Calib."X-Spalte".spalte_2;
               "FB_DROP_DB".zielRack.Position_Y := "DB_Referenzen".Calib."Y-Reihe".reihe_A;
           ELSIF "DB_Global".Order.Drop.rack = 'A3' THEN
               "FB_DROP_DB".zielRack.Position_X := "DB_Referenzen".Calib."X-Spalte".spalte_3;
               "FB_DROP_DB".zielRack.Position_Y := "DB_Referenzen".Calib."Y-Reihe".reihe_A;
           ELSIF "DB_Global".Order.Drop.rack = 'B1' THEN
               "FB_DROP_DB".zielRack.Position_X := "DB_Referenzen".Calib."X-Spalte".spalte_1;
               "FB_DROP_DB".zielRack.Position_Y := "DB_Referenzen".Calib."Y-Reihe".reihe_B;
           ELSIF "DB_Global".Order.Drop.rack = 'B2' THEN
               "FB_DROP_DB".zielRack.Position_X := "DB_Referenzen".Calib."X-Spalte".spalte_2;
               "FB_DROP_DB".zielRack.Position_Y := "DB_Referenzen".Calib."Y-Reihe".reihe_B;
           ELSIF "DB_Global".Order.Drop.rack = 'B3' THEN
               "FB_DROP_DB".zielRack.Position_X := "DB_Referenzen".Calib."X-Spalte".spalte_3;
               "FB_DROP_DB".zielRack.Position_Y := "DB_Referenzen".Calib."Y-Reihe".reihe_B;
           ELSIF "DB_Global".Order.Drop.rack = 'C1' THEN
               "FB_DROP_DB".zielRack.Position_X := "DB_Referenzen".Calib."X-Spalte".spalte_1;
               "FB_DROP_DB".zielRack.Position_Y := "DB_Referenzen".Calib."Y-Reihe".reihe_C;
           ELSIF "DB_Global".Order.Drop.rack = 'C2' THEN
               "FB_DROP_DB".zielRack.Position_X := "DB_Referenzen".Calib."X-Spalte".spalte_2;
               "FB_DROP_DB".zielRack.Position_Y := "DB_Referenzen".Calib."Y-Reihe".reihe_C;
           ELSIF "DB_Global".Order.Drop.rack = 'C3' THEN
               "FB_DROP_DB".zielRack.Position_X := "DB_Referenzen".Calib."X-Spalte".spalte_3;
               "FB_DROP_DB".zielRack.Position_Y := "DB_Referenzen".Calib."Y-Reihe".reihe_C;
           END_IF;
           #step := 31
           ;
       31: // Starte DROP 
           "FB_DROP_DB".finished := FALSE;
           "FB_DROP_DB".start := TRUE;
           #step := 32
           ;
       32: // Warte auf Finish
           IF "FB_DROP_DB".finished THEN
               #step := 33;
           END_IF
           ;
       33: // starte Referenzierung
           "DB_Global".DrehAchse.referenziert := FALSE;
           "DB_Global"."X-Achse".referenziert := FALSE;
           "DB_Global"."Y-Achse".referenziert := FALSE;
           #step := 34
           ;
       34: // warte auf ende Referenzierung
           IF "DB_Global".Referenziert THEN
               #step := 35;
           END_IF
           ;
       35: // bestätige erfolgreichen Abschluss 
           "DB_Global".Order.Drop.dropFinished := TRUE;
           "DB_Global".Order.Drop.dropAktiv := FALSE;
           "FB_DROP_DB".finished := FALSE;
           #step := 200
           ;

           // -------------------- ENDE DROP --------------------
       ELSE  // Statement section ELSE
           ;
   END_CASE;
END_REGION
END_FUNCTION_BLOCK

FUNCTION_BLOCK "FB_KALIBRIERE"   // FB5, FBD
{ S7_Optimized_Access := 'TRUE' }
VERSION : 0.1
   VAR
      fertig : Bool;
      "step" : DInt;
      "Timer" : TON_TIME;
      StartTimer : Bool;
      ZeitTimer : Time := T#1S;
   END_VAR
BEGIN

REGION Network 1 (SCL)
   CASE #step OF
       0: // Init

           IF "DB_Global".Order.Kalibriere.kalibAktiv THEN
               #step := 1;
           ELSE
               "DB_Global".Order.Kalibriere.DEFAULT := FALSE;
               "DB_Global".Order.Kalibriere.ANFAHREN := FALSE;
               "DB_Global".Order.Kalibriere.BEENDEN := FALSE;
               "DB_Global".Order.Park.PARK := FALSE;
               "DB_Global".Order.Park.parkAktiv := FALSE;
           END_IF
           ;
       1:  // Welche Steps

           IF "DB_Global".Order.Kalibriere.ANFAHREN THEN
               #step := 10;
               ;
           ELSIF "DB_Global".Order.Kalibriere.DEFAULT THEN
               #step := 20;
               ;
           ELSIF "DB_Global".Order.Kalibriere.BEENDEN THEN
               #step := 30;
               ;
           ELSIF "DB_Global".Order.Park.PARK THEN
               #step := 40;
               ;
           END_IF;

       10: // Die positionen Anfahren
           // Positionen übertragen
           "FB_Positionierung_DB".Achsen.X.sollPosition := "DB_Global".Order.Kalibriere.position_x;
           "FB_Positionierung_DB".Achsen.Y.sollPosition := "DB_Global".Order.Kalibriere.position_y;
           "FB_Positionierung_DB".Achsen.Dreh.sollPosition := "DB_Global".Order.Kalibriere.position_dreh;

           // positionierung Starten
           "FB_Positionierung_DB".finished := FALSE;
           "FB_Positionierung_DB".startPositionierung := TRUE;
           #step := 11;
           ;
       11: // warten auf Positionierung warten
           IF "FB_Positionierung_DB".finished THEN
               #step := 12;
           END_IF
           ;
       12: // Fertig
           "DB_Global".Order.Kalibriere.anfahrenBeendet := TRUE;
           "DB_Global".Order.Kalibriere.ANFAHREN := FALSE;
           #step := 13;
       13: // 
           #StartTimer := TRUE;
           IF #Timer.Q THEN
               #StartTimer := FALSE;
               "DB_Global".Order.Kalibriere.anfahrenBeendet := FALSE;
               #step := 1;
           END_IF
           ;
       20: // Auf Defaultwerte zurücksetzen

           "DB_Referenzen".Calib."Y-Reihe".reihe_A := "DB_Referenzen".Defaults."Y-Reihe".reihe_A;
           "DB_Referenzen".Calib."Y-Reihe".reihe_B := "DB_Referenzen".Defaults."Y-Reihe".reihe_B;
           "DB_Referenzen".Calib."Y-Reihe".reihe_C := "DB_Referenzen".Defaults."Y-Reihe".reihe_C;
           "DB_Referenzen".Calib."Y-Reihe".Offset := "DB_Referenzen".Defaults."Y-Reihe".Offset;

           "DB_Referenzen".Calib."X-Spalte".spalte_1 := "DB_Referenzen".Defaults."X-Spalte".spalte_1;
           "DB_Referenzen".Calib."X-Spalte".spalte_2 := "DB_Referenzen".Defaults."X-Spalte".spalte_2;
           "DB_Referenzen".Calib."X-Spalte".spalte_3 := "DB_Referenzen".Defaults."X-Spalte".spalte_3;

           "DB_Referenzen".Calib.Rampe.position_X := "DB_Referenzen".Defaults.Rampe.position_X;
           "DB_Referenzen".Calib.Rampe.position_Y := "DB_Referenzen".Defaults.Rampe.position_Y;
           "DB_Referenzen".Calib.Rampe.position_dreh := "DB_Referenzen".Defaults.Rampe.position_dreh;
           "DB_Referenzen".Calib.Rampe.offset := "DB_Referenzen".Defaults.Rampe.offset;

           "DB_Referenzen".Calib.FTS.Dreh := "DB_Referenzen".Defaults.FTS.Dreh;

           "DB_Referenzen".Calib.Limits.grenze_x_oben := "DB_Referenzen".Defaults.Limits.grenze_x_oben;
           "DB_Referenzen".Calib.Limits.grenze_x_unten := "DB_Referenzen".Defaults.Limits.grenze_x_unten;
           "DB_Referenzen".Calib.Limits.grenze_y_oben := "DB_Referenzen".Defaults.Limits.grenze_y_oben;
           "DB_Referenzen".Calib.Limits.grenze_y_unten := "DB_Referenzen".Defaults.Limits.grenze_y_unten;
           "DB_Referenzen".Calib.Limits.grenze_dreh_oben := "DB_Referenzen".Defaults.Limits.grenze_dreh_oben;
           "DB_Referenzen".Calib.Limits.grenze_dreh_unten := "DB_Referenzen".Defaults.Limits.grenze_dreh_unten;

           "DB_Referenzen".Calib.Zeiten.zeit_prozessende := "DB_Referenzen".Defaults.Zeiten.zeit_prozessende;
           "DB_Referenzen".Calib.Zeiten.zeit_saugerVentilAuf := "DB_Referenzen".Defaults.Zeiten.zeit_saugerVentilAuf;
           "DB_Referenzen".Calib.Zeiten.zeit_saugerVentilZu := "DB_Referenzen".Defaults.Zeiten.zeit_saugerVentilZu;
           "DB_Referenzen".Calib.Zeiten.zeit_kompressor := "DB_Referenzen".Defaults.Zeiten.zeit_kompressor;

           "DB_Referenzen".Calib.Park.position_x := "DB_Referenzen".Defaults.Park.position_x;
           "DB_Referenzen".Calib.Park.position_y := "DB_Referenzen".Defaults.Park.position_y;
           "DB_Referenzen".Calib.Park.position_dreh := "DB_Referenzen".Defaults.Park.position_dreh;

           "DB_Global".Order.Kalibriere.defaultBeendet:= TRUE;

           #step := 21;
       21: 
           "DB_Global".Order.Kalibriere.DEFAULT := FALSE;
           #StartTimer := TRUE;
           IF #Timer.Q THEN
               #StartTimer := FALSE;
               "DB_Global".Order.Kalibriere.defaultBeendet := FALSE;
               #step := 1;
           END_IF
           ;
       30: // Beenden
           #step := 31;
       31: // zurückfahren auf 0 
           // Positionen übertragen
           "FB_Positionierung_DB".Achsen.X.sollPosition := 0;
           "FB_Positionierung_DB".Achsen.Y.sollPosition := 0;
           "FB_Positionierung_DB".Achsen.Dreh.sollPosition := 0;

           // positionierung Starten
           "FB_Positionierung_DB".finished := FALSE;
           "FB_Positionierung_DB".startPositionierung := TRUE;
           #step := 32;
           ;
       32: // warten auf Positionierung warten
           IF "FB_Positionierung_DB".finished THEN
               #step := 33;
           END_IF
           ;
       33: // Fertig
           #fertig := TRUE;
           #StartTimer := TRUE;
           IF #Timer.Q THEN
               #StartTimer := FALSE;
               "DB_Global".Order.Kalibriere.BEENDEN := FALSE;
               #fertig := FALSE;
               #step := 0;
           END_IF
           ;
       40: // Park-Positionen als anfahr-Werte setzen
           "DB_Global".Order.Park.parkAktiv := TRUE;
           "DB_Global".Order.Kalibriere.position_x := "DB_Referenzen".Calib.Park.position_x;
           "DB_Global".Order.Kalibriere.position_y := "DB_Referenzen".Calib.Park.position_y;
           "DB_Global".Order.Kalibriere.position_dreh := "DB_Referenzen".Calib.Park.position_dreh;

           #step := 10; // direkt mit dem anfahren der gesetzten Positionen weitermachen
           ;
       ELSE  // Statement section ELSE
           ;
   END_CASE;
END_REGION

REGION Network 2
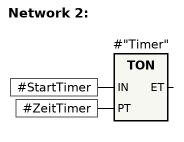
   #"Timer"(IN := #StartTimer, PT := #ZeitTimer);   // TON
END_REGION
END_FUNCTION_BLOCK

FUNCTION "FC_Verwaltung" : Void   // FC3, FBD
TITLE = Verwaltung
{ S7_Optimized_Access := 'TRUE' }
VERSION : 0.1
// Die High Speed Counter (HSC) sind hier definiert.
// 
// Die Pulsweitenmodulation (PWM), die für die richtige Ansteuerung der Encoder-Motoren notwendig sind werden hier.
BEGIN

REGION Network 1: DrehSauger Encoderwert
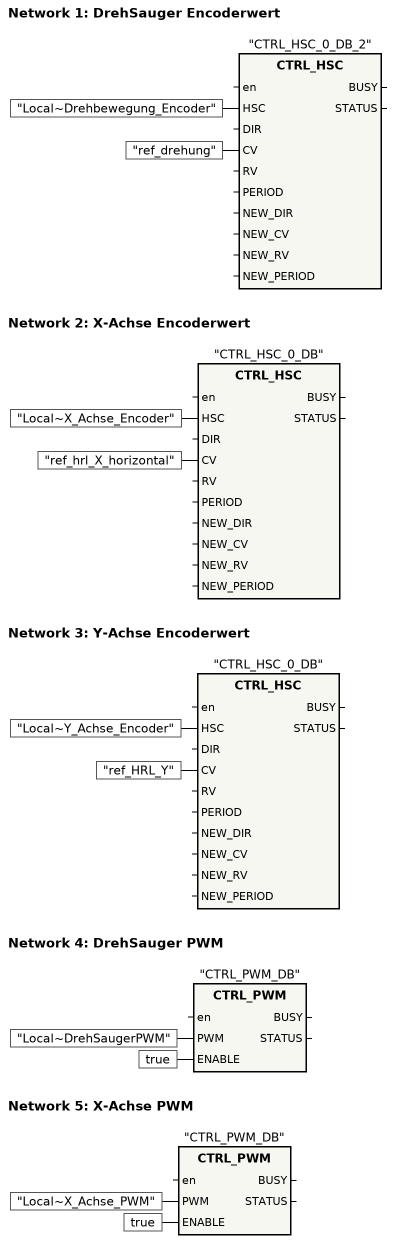
   "CTRL_HSC_0_DB_2"(HSC := "Local~Drehbewegung_Encoder", CV := "ref_drehung");   // CTRL_HSC
END_REGION

REGION Network 2: X-Achse Encoderwert
   "CTRL_HSC_0_DB"(HSC := "Local~X_Achse_Encoder", CV := "ref_hrl_X_horizontal");   // CTRL_HSC
END_REGION

REGION Network 3: Y-Achse Encoderwert
   "CTRL_HSC_0_DB"(HSC := "Local~Y_Achse_Encoder", CV := "ref_HRL_Y");   // CTRL_HSC
END_REGION

REGION Network 4: DrehSauger PWM
   "CTRL_PWM_DB"(PWM := "Local~DrehSaugerPWM", ENABLE := true);   // CTRL_PWM
END_REGION

REGION Network 5: X-Achse PWM
   "CTRL_PWM_DB"(PWM := "Local~X_Achse_PWM", ENABLE := true);   // CTRL_PWM
END_REGION

REGION Network 6: Y-Achse PWM
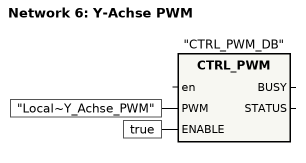
   "CTRL_PWM_DB"(PWM := "Local~Y_Achse_PWM", ENABLE := true);   // CTRL_PWM
END_REGION
END_FUNCTION

FUNCTION "FC_Referenzieren" : Void   // FC5, FBD
{ S7_Optimized_Access := 'TRUE' }
VERSION : 0.1
BEGIN

REGION Network 1: Power SaugerMotor
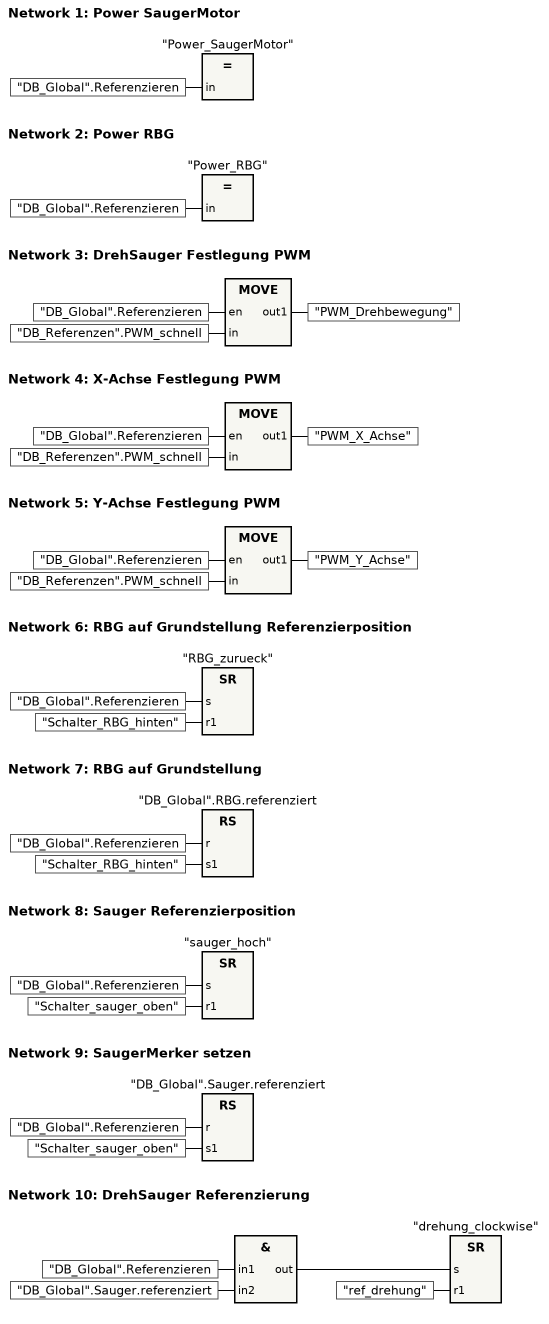
   "Power_SaugerMotor" := "DB_Global".Referenzieren;
END_REGION

REGION Network 2: Power RBG
   "Power_RBG" := "DB_Global".Referenzieren;
END_REGION

REGION Network 3: DrehSauger Festlegung PWM
   IF "DB_Global".Referenzieren THEN "PWM_Drehbewegung" := "DB_Referenzen".PWM_schnell; END_IF;
END_REGION

REGION Network 4: X-Achse Festlegung PWM
   IF "DB_Global".Referenzieren THEN "PWM_X_Achse" := "DB_Referenzen".PWM_schnell; END_IF;
END_REGION

REGION Network 5: Y-Achse Festlegung PWM
   IF "DB_Global".Referenzieren THEN "PWM_Y_Achse" := "DB_Referenzen".PWM_schnell; END_IF;
END_REGION

REGION Network 6: RBG auf Grundstellung Referenzierposition
   IF "DB_Global".Referenzieren THEN
       "RBG_zurueck" := TRUE;   // SR flip-flop
   END_IF;
   IF "Schalter_RBG_hinten" THEN "RBG_zurueck" := FALSE; END_IF;
END_REGION

REGION Network 7: RBG auf Grundstellung
   IF "DB_Global".Referenzieren THEN
       "DB_Global".RBG.referenziert := FALSE;   // RS flip-flop
   END_IF;
   IF "Schalter_RBG_hinten" THEN "DB_Global".RBG.referenziert := TRUE; END_IF;
END_REGION

REGION Network 8: Sauger Referenzierposition
   IF "DB_Global".Referenzieren THEN
       "sauger_hoch" := TRUE;   // SR flip-flop
   END_IF;
   IF "Schalter_sauger_oben" THEN "sauger_hoch" := FALSE; END_IF;
END_REGION

REGION Network 9: SaugerMerker setzen
   IF "DB_Global".Referenzieren THEN
       "DB_Global".Sauger.referenziert := FALSE;   // RS flip-flop
   END_IF;
   IF "Schalter_sauger_oben" THEN "DB_Global".Sauger.referenziert := TRUE; END_IF;
END_REGION

REGION Network 10: DrehSauger Referenzierung
   IF "DB_Global".Referenzieren AND "DB_Global".Sauger.referenziert THEN
       "drehung_clockwise" := TRUE;   // SR flip-flop
   END_IF;
   IF "ref_drehung" THEN "drehung_clockwise" := FALSE; END_IF;
END_REGION

REGION Network 11: DrehMerker setzen
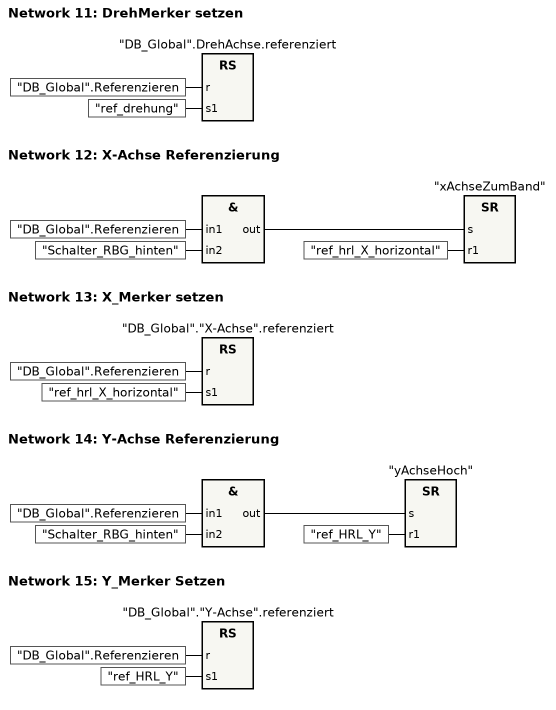
   IF "DB_Global".Referenzieren THEN
       "DB_Global".DrehAchse.referenziert := FALSE;   // RS flip-flop
   END_IF;
   IF "ref_drehung" THEN "DB_Global".DrehAchse.referenziert := TRUE; END_IF;
END_REGION

REGION Network 12: X-Achse Referenzierung
   IF "DB_Global".Referenzieren AND "Schalter_RBG_hinten" THEN
       "xAchseZumBand" := TRUE;   // SR flip-flop
   END_IF;
   IF "ref_hrl_X_horizontal" THEN "xAchseZumBand" := FALSE; END_IF;
END_REGION

REGION Network 13: X_Merker setzen
   IF "DB_Global".Referenzieren THEN
       "DB_Global"."X-Achse".referenziert := FALSE;   // RS flip-flop
   END_IF;
   IF "ref_hrl_X_horizontal" THEN "DB_Global"."X-Achse".referenziert := TRUE; END_IF;
END_REGION

REGION Network 14: Y-Achse Referenzierung
   IF "DB_Global".Referenzieren AND "Schalter_RBG_hinten" THEN
       "yAchseHoch" := TRUE;   // SR flip-flop
   END_IF;
   IF "ref_HRL_Y" THEN "yAchseHoch" := FALSE; END_IF;
END_REGION

REGION Network 15: Y_Merker Setzen
   IF "DB_Global".Referenzieren THEN
       "DB_Global"."Y-Achse".referenziert := FALSE;   // RS flip-flop
   END_IF;
   IF "ref_HRL_Y" THEN "DB_Global"."Y-Achse".referenziert := TRUE; END_IF;
END_REGION
END_FUNCTION

ORGANIZATION_BLOCK "Main"   // OB1, FBD, ProgramCycle
{ S7_Optimized_Access := 'TRUE' }
VERSION : 0.1
   VAR_INPUT
      Initial_Call : Bool;
      Remanence : Bool;
   END_VAR
   VAR_TEMP   // added for the SCL form of the ladder/FBD networks
      _w1 : Bool;
   END_VAR
BEGIN

REGION Network 1: Bausteinaufruf FC3 Verwaltung
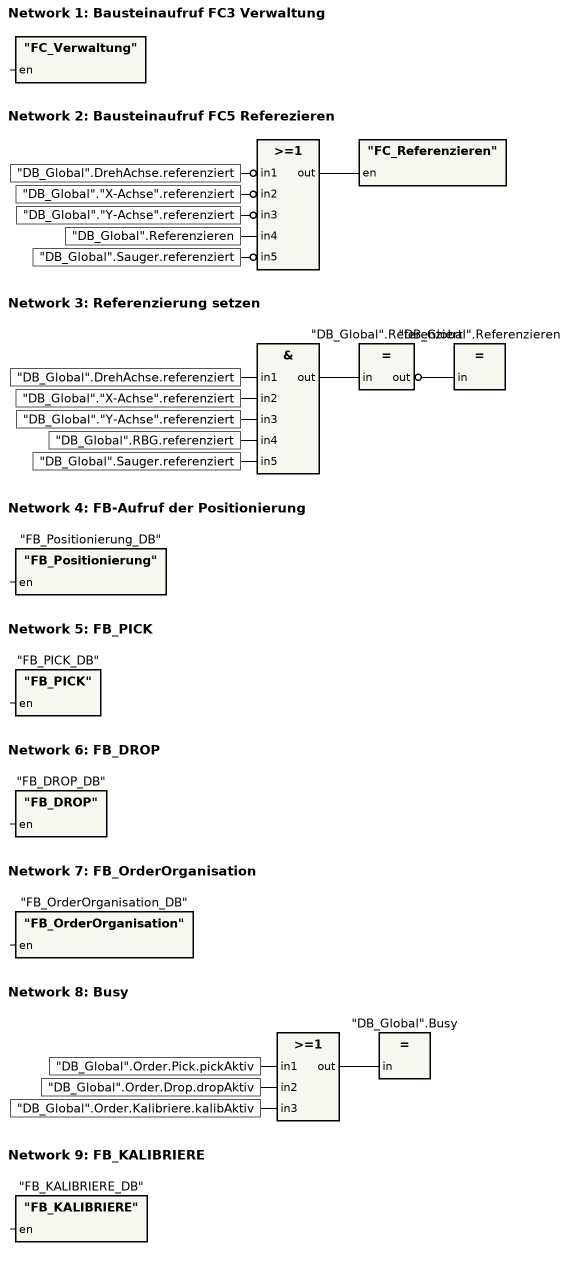
   "FC_Verwaltung"();
END_REGION

REGION Network 2: Bausteinaufruf FC5 Referezieren
   IF NOT "DB_Global".DrehAchse.referenziert OR NOT "DB_Global"."X-Achse".referenziert OR NOT "DB_Global"."Y-Achse".referenziert OR "DB_Global".Referenzieren OR NOT "DB_Global".Sauger.referenziert THEN
       "FC_Referenzieren"();
   END_IF;
END_REGION

REGION Network 3: Referenzierung setzen
   #_w1 := "DB_Global".DrehAchse.referenziert AND "DB_Global"."X-Achse".referenziert AND "DB_Global"."Y-Achse".referenziert AND "DB_Global".RBG.referenziert AND "DB_Global".Sauger.referenziert;
   "DB_Global".Referenziert := #_w1;
   "DB_Global".Referenzieren := NOT #_w1;
END_REGION

REGION Network 4: FB-Aufruf der Positionierung
   "FB_Positionierung_DB"();   // "FB_Positionierung"
END_REGION

REGION Network 5: FB_PICK
   "FB_PICK_DB"();   // "FB_PICK"
END_REGION

REGION Network 6: FB_DROP
   "FB_DROP_DB"();   // "FB_DROP"
END_REGION

REGION Network 7: FB_OrderOrganisation
   "FB_OrderOrganisation_DB"();   // "FB_OrderOrganisation"
END_REGION

REGION Network 8: Busy
   "DB_Global".Busy := "DB_Global".Order.Pick.pickAktiv OR "DB_Global".Order.Drop.dropAktiv OR "DB_Global".Order.Kalibriere.kalibAktiv;
END_REGION

REGION Network 9: FB_KALIBRIERE
   "FB_KALIBRIERE_DB"();   // "FB_KALIBRIERE"
END_REGION
END_ORGANIZATION_BLOCK

// folder: EncoderMoves

FUNCTION_BLOCK "FB_Positionierung"   // FB1, FBD
TITLE = Positionierung
{ S7_Optimized_Access := 'TRUE' }
VERSION : 0.1
// Der Baustein muss im Main dauerhaft an sein um richtig zu funktionieren
// 
// Bevor die Variable "startPositionierung" TRUE und "finished" FALSE gesetzt werden.
// Die "Sollpositionen" sind genauso müssen auch übertragen worden sein bevor die startPositionierung TRUE gesetzt wird.
// 
// "finished" wird vom Baustein wieder TRUE gesetzt wenn, alle 3 Achsen die Position erreicht haben.
   VAR
      startPositionierung : Bool;
      working : Bool;
      finished : Bool;
      Achsen : Struct
         X : Struct
            sollPosition : DInt;
            start : Bool;
            positionErreicht : Bool;
         END_STRUCT;
         Y : Struct
            sollPosition : DInt;
            start : Bool;
            positionErreicht : Bool;
         END_STRUCT;
         Dreh : Struct
            sollPosition : DInt;
            start : Bool;
            positionErreicht : Bool;
         END_STRUCT;
      END_STRUCT;
      "step" : DInt;
      zuGroßX : Bool;
      zuKleinX : Bool;
      zuGroßY : Bool;
      zuKleinY : Bool;
      zuGroßDreh : Bool;
      zuKleinDreh : Bool;
   END_VAR
BEGIN

REGION Network 1 (SCL): Schrittkette
   CASE #step OF
       0:  // Start Positionierung
           IF #startPositionierung AND NOT #working THEN
               #startPositionierung := FALSE;
               #working := TRUE;
               #step := 1;
           END_IF
           ;
       1: // check ob variablen außerhalb der Limits ist
           // X-Achse
           IF #zuGroßX THEN
               #Achsen.X.sollPosition := "DB_Referenzen".Calib.Limits.grenze_x_oben
               ;
           ELSIF #zuKleinX THEN
               #Achsen.X.sollPosition := "DB_Referenzen".Calib.Limits.grenze_x_unten
               ;
           END_IF
           ;
           // Y-Achse
           IF #zuGroßY THEN
               #Achsen.Y.sollPosition := "DB_Referenzen".Calib.Limits.grenze_y_oben
               ;
           ELSIF #zuKleinY THEN
               #Achsen.Y.sollPosition := "DB_Referenzen".Calib.Limits.grenze_y_unten
               ;
           END_IF
           ;
           // DREH-Achse
           IF #zuGroßDreh THEN
               #Achsen.Dreh.sollPosition := "DB_Referenzen".Calib.Limits.grenze_dreh_oben
               ;
           ELSIF #zuKleinDreh THEN
               #Achsen.Dreh.sollPosition := "DB_Referenzen".Calib.Limits.grenze_dreh_unten
               ;
           END_IF
           ;
           #step := 2;
       2:  // Starte Achsen
           #Achsen.X.positionErreicht := FALSE;
           #Achsen.Y.positionErreicht := FALSE;
           #Achsen.Dreh.positionErreicht := FALSE;

           #Achsen.X.start := TRUE;
           #Achsen.Y.start := TRUE;
           #Achsen.Dreh.start := TRUE;

           #step := 10;

       10:  // Stoppe Achsen
           IF #Achsen.X.positionErreicht THEN
               #Achsen.X.start := FALSE;
           END_IF;

           IF #Achsen.Y.positionErreicht THEN
               #Achsen.Y.start := FALSE;
           END_IF;

           IF #Achsen.Dreh.positionErreicht THEN
               #Achsen.Dreh.start := FALSE;
           END_IF;

           IF #Achsen.X.positionErreicht AND #Achsen.Y.positionErreicht AND #Achsen.Dreh.positionErreicht THEN
               #step := 20;
           END_IF
           ;
       20: // 
           #working := FALSE;
           #finished := TRUE;
           #step := 0
           ;
       ELSE  // Statement section ELSE
           ;
   END_CASE;
END_REGION

REGION Network 2: Positionierung X
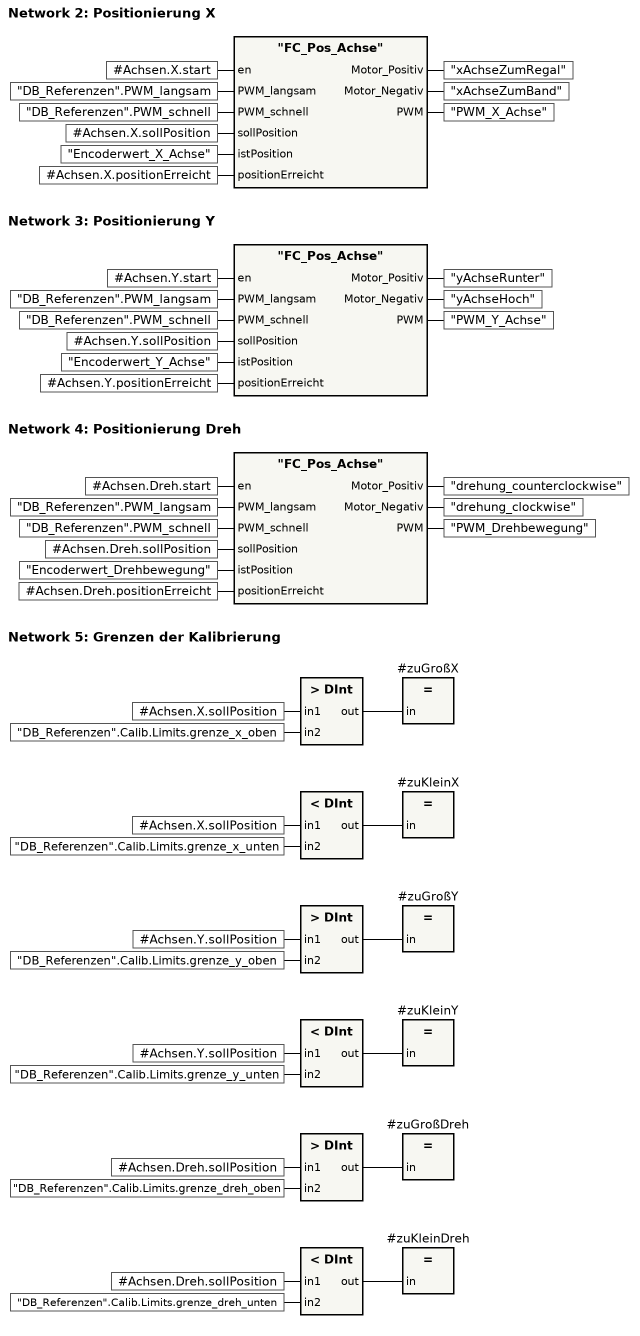
   IF #Achsen.X.start THEN
       "FC_Pos_Achse"(PWM_langsam := "DB_Referenzen".PWM_langsam,
                      PWM_schnell := "DB_Referenzen".PWM_schnell,
                      sollPosition := #Achsen.X.sollPosition,
                      istPosition := "Encoderwert_X_Achse",
                      positionErreicht := #Achsen.X.positionErreicht,
                      Motor_Positiv => "xAchseZumRegal",
                      Motor_Negativ => "xAchseZumBand",
                      PWM => "PWM_X_Achse");
   END_IF;
END_REGION

REGION Network 3: Positionierung Y
   IF #Achsen.Y.start THEN
       "FC_Pos_Achse"(PWM_langsam := "DB_Referenzen".PWM_langsam,
                      PWM_schnell := "DB_Referenzen".PWM_schnell,
                      sollPosition := #Achsen.Y.sollPosition,
                      istPosition := "Encoderwert_Y_Achse",
                      positionErreicht := #Achsen.Y.positionErreicht,
                      Motor_Positiv => "yAchseRunter",
                      Motor_Negativ => "yAchseHoch",
                      PWM => "PWM_Y_Achse");
   END_IF;
END_REGION

REGION Network 4: Positionierung Dreh
   IF #Achsen.Dreh.start THEN
       "FC_Pos_Achse"(PWM_langsam := "DB_Referenzen".PWM_langsam,
                      PWM_schnell := "DB_Referenzen".PWM_schnell,
                      sollPosition := #Achsen.Dreh.sollPosition,
                      istPosition := "Encoderwert_Drehbewegung",
                      positionErreicht := #Achsen.Dreh.positionErreicht,
                      Motor_Positiv => "drehung_counterclockwise",
                      Motor_Negativ => "drehung_clockwise",
                      PWM => "PWM_Drehbewegung");
   END_IF;
END_REGION

REGION Network 5: Grenzen der Kalibrierung
   #zuGroßX := #Achsen.X.sollPosition > "DB_Referenzen".Calib.Limits.grenze_x_oben;
   #zuKleinX := #Achsen.X.sollPosition < "DB_Referenzen".Calib.Limits.grenze_x_unten;
   #zuGroßY := #Achsen.Y.sollPosition > "DB_Referenzen".Calib.Limits.grenze_y_oben;
   #zuKleinY := #Achsen.Y.sollPosition < "DB_Referenzen".Calib.Limits.grenze_y_unten;
   #zuGroßDreh := #Achsen.Dreh.sollPosition > "DB_Referenzen".Calib.Limits.grenze_dreh_oben;
   #zuKleinDreh := #Achsen.Dreh.sollPosition < "DB_Referenzen".Calib.Limits.grenze_dreh_unten;
END_REGION
END_FUNCTION_BLOCK

FUNCTION "FC_Pos_Achse" : Void   // FC9, FBD
{ S7_Optimized_Access := 'TRUE' }
VERSION : 0.1
   VAR_INPUT
      PWM_langsam : DInt;
      PWM_schnell : DInt;
      sollPosition : DInt;
      istPosition : DInt;
   END_VAR
   VAR_OUTPUT
      Motor_Positiv : Bool;
      Motor_Negativ : Bool;
      PWM : DInt;
   END_VAR
   VAR_IN_OUT
      positionErreicht : Bool;
   END_VAR
   VAR_TEMP
      langsamOben : DInt;
      langsamUnten : DInt;
      grenzeOben : DInt;
      grenzeUnten : DInt;
   END_VAR
   VAR_TEMP   // added for the SCL form of the ladder/FBD networks
      _w1 : Bool;
   END_VAR
BEGIN

REGION Network 1: Berechne Grenzen X
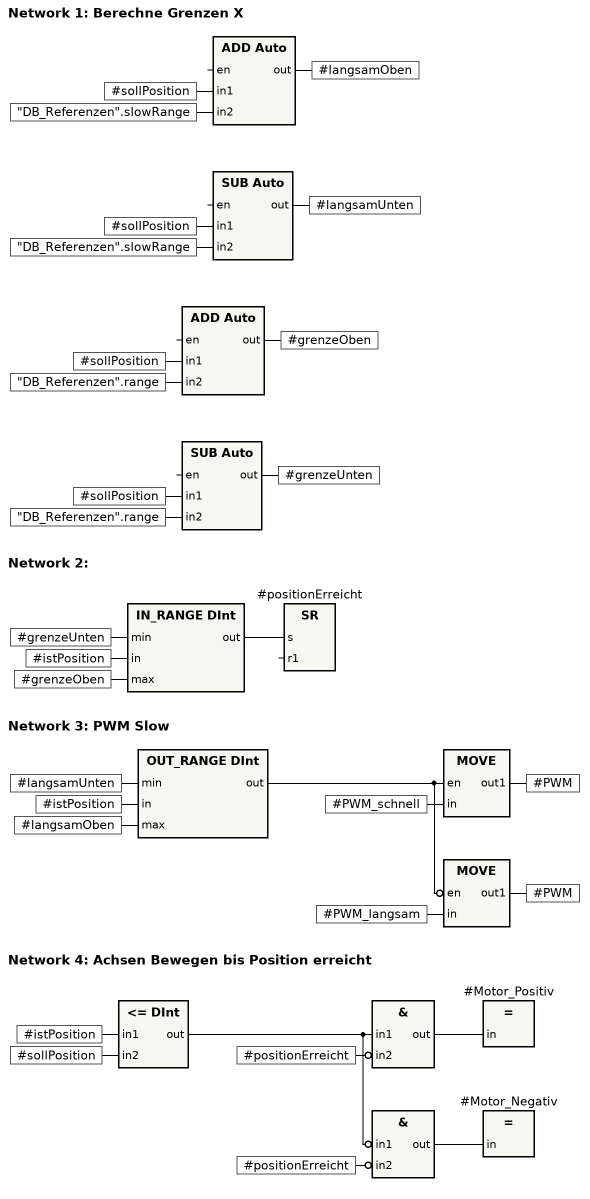
   #langsamOben := #sollPosition + "DB_Referenzen".slowRange;
   #langsamUnten := #sollPosition - "DB_Referenzen".slowRange;
   #grenzeOben := #sollPosition + "DB_Referenzen".range;
   #grenzeUnten := #sollPosition - "DB_Referenzen".range;
END_REGION

REGION Network 2
   IF (#grenzeUnten <= #istPosition) AND (#istPosition <= #grenzeOben) THEN
       #positionErreicht := TRUE;   // SR flip-flop
   END_IF;
END_REGION

REGION Network 3: PWM Slow
   #_w1 := (#istPosition < #langsamUnten) OR (#istPosition > #langsamOben);
   IF #_w1 THEN #PWM := #PWM_schnell; END_IF;
   IF NOT #_w1 THEN #PWM := #PWM_langsam; END_IF;
END_REGION

REGION Network 4: Achsen Bewegen bis Position erreicht
   #_w1 := #istPosition <= #sollPosition;
   #Motor_Positiv := #_w1 AND NOT #positionErreicht;
   #Motor_Negativ := NOT #_w1 AND NOT #positionErreicht;
END_REGION
END_FUNCTION